// SIMATIC S7-200 project (STEP 7-Micro/WIN), CPU 224XP REL 02.00

ORGANIZATION_BLOCK 主程序:OB1
TITLE=彩灯控制
// 8位彩灯的追灯控制程序。
// 要求可以改变追灯的花样
// 能够改变彩灯移位速度
// 能够改变彩灯移动方向
BEGIN
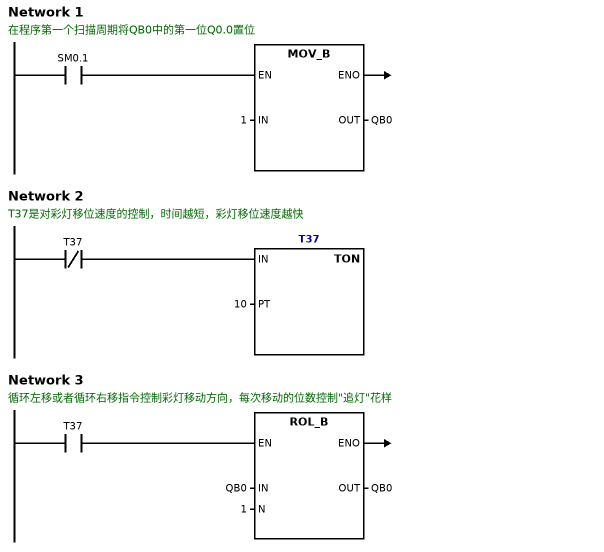
Network 1
// 在程序第一个扫描周期将QB0中的第一位Q0.0置位
LD     SM0.1
MOVB   1, QB0
Network 2
// T37是对彩灯移位速度的控制，时间越短，彩灯移位速度越快
LDN    T37
TON    T37, 10
Network 3
// 循环左移或者循环右移指令控制彩灯移动方向，每次移动的位数控制"追灯"花样
LD     T37
RLB    QB0, 1
END_ORGANIZATION_BLOCK
